Fanuc KAREL source: kt00976.KL

-- PROVISIONAL review KL for V770-1; original PC SHA256 31504037de854a4c027ce3c5a9623c5989b53500145de457d5500556a6b6b04f
-- Incomplete behavior may be omitted. Consult companion uncertainty JSON. Do not deploy.
PROGRAM KT00976
%NOLOCKGROUP
BEGIN
  -- UNRESOLVED_PC offsets 5-12; opcodes 9C,23
  -- UNRESOLVED_PC offsets 17-25; opcodes 3F,75
  -- UNRESOLVED_PC offsets 30-43; opcodes 3F,75
  -- UNRESOLVED_PC offsets 48-86; opcodes 27,22,22,2A,22,2A,22,22,B0
  -- UNRESOLVED_PC offsets 91-95; opcodes 7F
END KT00976
